FUNCTION_BLOCK FB_ASDAB3_RTU EXTENDS FB_ModbusSlaveRtu
VAR
	eState : E_ASDAB3_State;
	bBusy : BOOL;
	bInit : BOOL;
	bInited : BOOL;
	bActive : BOOL;
	bIsStop : BOOL;
	bHomed : BOOL;
	bHome : BOOL;
	bReset : BOOL;
	bAlarm : BOOL;
	bAbort : BOOL;
	bMoveAbsolute : BOOL;
	eStatus : E_ASDAB3_Status;
	fPositionFB : LREAL;
	fVelocityFB : LREAL;								// Unit: rpm
	fTorqueFB : LREAL;									// %
	fPositionCMD : LREAL;	
	fHomePosition : LREAL;
	nFaultCode	: INT;
	TempData_w2di	: ARRAY[0..2] OF U_Word2Dint;
	uPositionCmd : U_Word2Dint;
	wDoStatus : WORD;
	//tonClock : TON;
END_VAR

SUPER^();
bActive := eState>=IPRO_READY_INITIALIZED;
bError := bModbusError OR nFaultCode<>0;
CASE eState OF
	asdab3_INITIALIZING..asdab3_RESET_DONE, asdab3_ABORTING:
		tonConfirmReallyError(
			IN := bError OR bModbusError,
			PT := timeConfirmReallyError,
			Q => bReallyError 
		);
END_CASE
StateMachine();

PROPERTY Active : bool
GET
Active := bActive;
END_GET
END_PROPERTY

PROPERTY Busy : bool
GET
Busy := bBusy;
END_GET
END_PROPERTY

METHOD Convert : BOOL
VAR_INPUT
	iRegionNo	:	INT;
	pReadData	:	POINTER TO word;
END_VAR

CASE iRegionNo OF 
	0:	// positionFB, SpeedFB, and Torque FB
		TempData_w2di[0].iWord[0] := pReadData[0];
		TempData_w2di[0].iWord[1] := pReadData[1];
		TempData_w2di[1].iWord[0] := pReadData[2];
		TempData_w2di[1].iWord[1] := pReadData[3];
		TempData_w2di[2].iWord[0] := pReadData[4];
		TempData_w2di[2].iWord[1] := pReadData[5];
		fPositionFB := DINT_TO_LREAL(TempData_w2di[0].idInt);
		fVelocityFB := 0.1*DINT_TO_LREAL(TempData_w2di[1].idInt);
		fTorqueFB := 0.1*DINT_TO_LREAL(TempData_w2di[2].idInt);
		
	1:	// DO Register
		wDoStatus := pReadData[0];
		IF ModbusErrorID = MODBUSERROR_NO_RESPONSE THEN
			eStatus := ASDAB3_STATUS_NOT_RESPOND;
		ELSIF wDoStatus.6 THEN
			eStatus := ASDAB3_STATUS_FAULT;
		ELSIF wDoStatus.0 AND NOT wDoStatus.1 THEN
			eStatus := ASDAB3_STATUS_READY;
		ELSIF wDoStatus.1 THEN
			eStatus := ASDAB3_STATUS_ACTIVE;
		END_IF
		bHomed := wDoStatus.8;
	2:
		nFaultCode := WORD_TO_INT(pReadData[0]);
	
	
END_CASE
END_METHOD

PROPERTY ErrorID : REFERENCE TO INT
GET
errorid ref= nFaultCode;
END_GET
END_PROPERTY

PROPERTY Homed : bool
GET
Homed := bHomed;
END_GET
END_PROPERTY

PROPERTY InPosition : bool
GET
Inposition := F_CheckInRange(
					lrHighLimit := fPositionCMD+5,
					lrLowLimit := fPositionCMD-5,
					lrValue := fPositionFB
				);
END_GET
END_PROPERTY

PROPERTY IsStop : bool
GET
IsStop := bIsStop;
END_GET
END_PROPERTY

METHOD MR_Abort : BOOL // THIS IS REQUEST ABORT. => ACTIVE = False
IF eState >= ASDAB3_INITIALIZING THEN
	bAbort := TRUE;
	MR_Abort := FALSE;
	bBusy := TRUE;
	eState := ASDAB3_ABORTING;
ELSIF eState = ASDAB3_UNINITIALIZED THEN
	bAbort := FALSE;
	MR_Abort := TRUE;
	bBusy := False;
END_IF
END_METHOD

METHOD MR_Home : BOOL	// use for homing only, not use for move to position.
VAR_INPUT
	lrHomePosition : LREAL;		//	Absolute reference position to which the axis is set after homing.
END_VAR
IF eState = ASDAB3_IDLE AND NOT bHomed THEN 
	bHome := TRUE;
	bBusy := TRUE;  
	MR_Home := FALSE;
 	eState := ASDAB3_HOME;
	fHomePosition := lrHomePosition;
	
ELSIF eState = ASDAB3_HOME_DONE THEN
	bHome := FALSE;
	bBusy := FALSE;
	MR_Home := TRUE;
END_IF
END_METHOD

METHOD MR_Init : BOOL
IF eState = ASDAB3_UNINITIALIZED THEN
	bInit := TRUE;
	bInited := FALSE;
	bBusy := TRUE;
	MR_Init := FALSE;
	eState := ASDAB3_INITIALIZING;
ELSIF eState = ASDAB3_READY_INITIALIZED THEN
	bInited := True;
	bInit := FALSE;
	bBusy := FALSE;
	MR_Init := TRUE;
	
END_IF
END_METHOD

METHOD MR_MoveAbsolute : BOOL // control mode must have Position Mode
VAR_INPUT
	lrAbsolutePosition : LREAL;
END_VAR
IF eState = ASDAB3_IDLE 
AND NOT F_CheckInRange(
			lrHighLimit := fPositionFB+5,
			lrLowLimit := fPositionfb-5,
			lrValue := lrAbsolutePosition
		)										
THEN
	fPositionCMD := lrAbsolutePosition;
	MR_MoveAbsolute := FALSE;
	bBusy := TRUE;
	bMoveAbsolute := TRUE;
	eState := ASDAB3_MOVE_ABSOLUTE;

ELSIF eState = ASDAB3_MOVE_ABSOLUTE_DONE THEN
	bBusy := FALSE;
	bMoveAbsolute := FALSE;
	MR_MoveAbsolute := TRUE;
END_IF
END_METHOD

METHOD MR_Reset : BOOL// can't not use this method because i didn't find way to reset
IF bError AND eState<>ASDAB3_RESET THEN
	bReset := TRUE;
	MR_Reset := FALSE;
	eState := ASDAB3_RESET;
ELSIF eState = ASDAB3_RESET_DONE THEN
	bReset := FALSE;
	MR_Reset := TRUE;	
END_IF
END_METHOD

METHOD PROTECTED MS_Aborting// still remain all the params set before init
VAR_INPUT
END_VAR
arrAddressWrite[1][2] := 2#0;
fPositionCMD := 0;
IF NOT wDoStatus.1 THEN
	eState := ASDAB3_UNINITIALIZED;
END_IF
END_METHOD

METHOD PROTECTED MS_Home
VAR_INPUT
END_VAR
arrAddressWrite[1][2].3 := TRUE;
IF bHomed THEN
	eState := ASDAB3_HOME_DONE;
END_IF
END_METHOD

METHOD PROTECTED  MS_HomeDone
VAR_INPUT
END_VAR
IF NOT bHome THEN
	eState := ASDAB3_IDLE;
END_IF
END_METHOD

METHOD PROTECTED MS_Idle
VAR_INPUT
END_VAR
arrAddressWrite[1][2].3 := FALSE;
arrAddressWrite[1][2].2 := FALSE;
bBusy := false;
END_METHOD

METHOD PROTECTED MS_Initializing
VAR_INPUT
END_VAR
arrAddressWrite[1][2] := 2#11;
IF eStatus = ASDAB3_STATUS_ACTIVE THEN
	eState := ASDAB3_READY_INITIALIZED;
END_IF
END_METHOD

METHOD PROTECTED MS_MoveAbsolute
VAR_INPUT
END_VAR
uPositionCmd.idInt := LREAL_TO_DINT(fPositionCMD);
arrAddressWrite[0][2] := uPositionCmd.iWord[0];
arrAddressWrite[0][3] := uPositionCmd.iWord[1];
arrAddressWrite[1][2].2 := TRUE;
IF InPosition THEN
	estate := ASDAB3_MOVE_ABSOLUTE_DONE;
END_IF
END_METHOD

METHOD PROTECTED MS_MoveAbsoluteDone
VAR_INPUT
END_VAR
IF NOT bMoveAbsolute THEN
	estate := ASDAB3_IDLE;
END_IF
END_METHOD

METHOD PROTECTED MS_ReadyInitialized
VAR_INPUT
END_VAR
arrAddressWrite[1][2] := 2#01;
IF NOT bInit THEN
	eState := ASDAB3_IDLE;
END_IF
END_METHOD

METHOD PROTECTED MS_Reset
VAR_INPUT
END_VAR
arrAddressWrite[1][2].1 := NOT arrAddressWrite[1][2].1;
IF NOT bError THEN
	estate := ASDAB3_RESET_DONE;
END_IF
END_METHOD

METHOD PROTECTED MS_ResetDone
VAR_INPUT
END_VAR
IF NOT bReset THEN
	eState := ASDAB3_IDLE;
END_IF
END_METHOD

METHOD PROTECTED MS_Uninitalized
VAR_INPUT
END_VAR
bBusy := FALSE;
// Read
arrAddressRead[0][0] := 16#12;	// monitoring position, speed, torque : P0.009
arrAddressRead[0][1] := 6;
arrAddressRead[0][2] := E_ModbusFunction.ReadHoldingRegisters;

arrAddressRead[1][0] := 16#5C; // Regiter Output: P0.046
arrAddressRead[1][1] := 1;
arrAddressRead[1][2] := E_ModbusFunction.ReadHoldingRegisters;

arrAddressRead[2][0] := 16#02; // errorID: P0.001
arrAddressRead[2][1] := 1;
arrAddressRead[2][2] := E_ModbusFunction.ReadHoldingRegisters;
iNumAddRegionRead := 3;

// write
arrAddressWrite[0][0] := 16#706; // Position cmd PR51 data
arrAddressWrite[0][1] := 2;
arrAddressWrite[0][2] := 0;
arrAddressWrite[0][10]	:= E_ModbusFunction.WriteMultipleRegisters;
(*	// DI register cmd:
	bit1: On : level Active
	bit2: reset alarm : rise trig
	bit3: execute run abs position
*)
arrAddressWrite[1][0] := 16#40E;
arrAddressWrite[1][1] := 1;
arrAddressWrite[1][2] := 0;
arrAddressWrite[1][10] := E_ModbusFunction.WriteSingleRegister;

arrAddressWrite[2][0] := 16#30C;	//P3.006 Digital input (DI) control switch
arrAddressWrite[2][1] := 1;
arrAddressWrite[2][2] := 16#1FFF;	//never change this value
arrAddressWrite[2][10] := E_ModbusFunction.WriteSingleRegister;

iNumAddRegionWrite := 3;
END_METHOD

PROPERTY PositionCmd : lreal
GET
PositionCmd := fPositionCMD;
END_GET
END_PROPERTY

METHOD PROTECTED StateMachine
VAR_INPUT
END_VAR
CASE eState OF
	ASDAB3_UNINITIALIZED :
		MS_Uninitalized();
		
	ASDAB3_INITIALIZING	:
		MS_Initializing();
		
	ASDAB3_READY_INITIALIZED :
		MS_ReadyInitialized();
		
	ASDAB3_IDLE	:
		MS_Idle();
		
	ASDAB3_MOVE_ABSOLUTE :
		MS_MoveAbsolute();
		
	ASDAB3_MOVE_ABSOLUTE_DONE :
		MS_MoveAbsoluteDone();
		
	ASDAB3_HOME:
		MS_Home();
		
	ASDAB3_HOME_DONE:
		MS_HomeDone();
	
	ASDAB3_RESET :
		MS_Reset();
		
	ASDAB3_RESET_DONE :
		MS_ResetDone();
		
	ASDAB3_ABORTING :
		MS_Aborting();
END_CASE
END_METHOD

END_FUNCTION_BLOCK

(* stored: Version 1.1.0.1, ProductVersion 3.1.4024.12
   POU FB_ASDAB3_RTU: Id {7bdd2ce4-5f9a-4631-959f-df0649514377}, SpecialFunc None
   Folder MR: Id {944ec9b4-8025-4605-ab1b-a15596047c6c}
   Folder MS: Id {bcb77bc9-36f9-4c14-ad25-95db4d61ba13}
   Folder Status: Id {ca1a44a3-914d-4ebb-b2d7-0aa2d4303451}
   Property Active: Id {ce5ec9f4-b294-43a2-a99e-72c65be75d32}
   Get Get: Id {924b0c43-4c58-47a4-9386-2d1182edf158}
   Property Busy: Id {18069665-9822-4578-a5e5-cb85a412bc2f}
   Get Get: Id {08a27e36-96ca-4f44-bdb4-9982c2e145fb}
   Method Convert: Id {c2c16085-ade9-48b8-9689-ed8cdf970e8d}
   Property ErrorID: Id {42de6558-78de-4dd3-bf04-5aacd5e26460}
   Get Get: Id {0f07ec2d-6c61-47bd-ae54-7377bde8a6a8}
   Property Homed: Id {af3ac53b-61f1-4d70-b085-5a8abd96aeca}
   Get Get: Id {d8b09f81-e1b8-4f7f-a263-47d049fe977a}
   Property InPosition: Id {88018cac-97af-4b1b-8f48-7ac2c904444f}
   Get Get: Id {4efaf9db-0bbe-40f9-990c-06372fb23ff5}
   Property IsStop: Id {45e2adc2-7c16-485a-b88c-85de616b1808}
   Get Get: Id {c37099d5-16ab-437e-92b9-1f4b95eda5f5}
   Method MR_Abort: Id {9915d01b-bbd3-4354-a629-9317fc233e21}
   Method MR_Home: Id {6eadc91d-8091-4708-9949-c97556344482}
   Method MR_Init: Id {7ca5025e-e8bb-4736-82b2-04545a0909fd}
   Method MR_MoveAbsolute: Id {87f73bf7-8dac-4507-a8cb-8fca6887c83c}
   Method MR_Reset: Id {c693223d-4977-4b6e-826e-480173adf595}
   Method MS_Aborting: Id {088a2ebc-58b1-4f2c-be44-14f0b7dccc09}
   Method MS_Home: Id {ebc03257-76f2-4a05-acfc-20baa18bb82e}
   Method MS_HomeDone: Id {8ec539d1-139b-4888-9a5d-f6860065708a}
   Method MS_Idle: Id {3f833b86-9014-4120-8cfa-25f3d00f7dc7}
   Method MS_Initializing: Id {562d926a-91da-4ef7-88ad-cac4d8dd4f76}
   Method MS_MoveAbsolute: Id {ce45af5c-d840-4ade-b299-c6b6e376d6d0}
   Method MS_MoveAbsoluteDone: Id {744f3b1f-cfe4-47c9-9fa1-86f4952b3bfe}
   Method MS_ReadyInitialized: Id {464b8d82-5009-4168-a158-6cbabb711e39}
   Method MS_Reset: Id {c6a785e2-c413-4c99-b762-e02831f57fae}
   Method MS_ResetDone: Id {38ccce8c-e844-4455-8a5f-e24ff30b51db}
   Method MS_Uninitalized: Id {4fa74425-b155-4722-8999-3c8f5d75d7b4}
   Property PositionCmd: Id {9abeab55-b77c-49ff-ab6e-596ba093758f}
   Get Get: Id {84e83cd0-56af-47cb-80d2-4bf661192527}
   Method StateMachine: Id {d7c30c34-6f72-4195-b9ee-9a5312f00a8f} *)
